// TIA Portal V20 export
DATA_BLOCK "GLOBAL_DRIVE_HMI_IF_DB"   // DB203
{ S7_Optimized_Access := 'TRUE' }
AUTHOR : Tesla
FAMILY : Drive
VERSION : 1.0
// stored: AutoNumber false, MemoryReserve 100
   VAR RETAIN
      Drive : Array[0.."No_Drives"] of "DRIVE_HMI_UDT";
   END_VAR
BEGIN
END_DATA_BLOCK
